// MajorComponents/FB_BPRequestor
(* BP Requestor
Elevates the BP request from an arbiter to PMPS_GVL.stRequestedBP
*)
FUNCTION_BLOCK FB_BPRequestor IMPLEMENTS I_HigherAuthority
VAR_INPUT
END_VAR
VAR_OUTPUT
    q_ReqBP : ST_BeamParams; // Arbitrated BP
END_VAR
VAR_IN_OUT
    Arbiter : FB_Arbiter;
    //FFO : FB_HardwareFFOutput;
END_VAR
VAR
    ReqBP : ST_BeamParams;
    nCohort : ULINT; // Current cohort, inc. 1 cycle after IO is updated
    nRequestCohort : ULINT; // Cohort number recorded at the time of the request.
END_VAR

Arbiter.ElevateRequest(THIS^); // Executes arbitration and retrieves ReqBP

IF nRequestCohort >= nCohort THEN
    // Update requested BP set
    q_ReqBP := ReqBP;
    // Note: we may do more here someday... perhaps all of the output control
    // will reside in here, and be solely controlled by this block. For now
    // I am going to adopt a flat management structure.
    // Start a new cohort
    nCohort := nCohort + 1;
END_IF

// Returns true when outputs to MPS are updated
METHOD CheckRequest : BOOL
VAR_INPUT
	nReqID	: DWORD;
END_VAR
VAR_INST
    xFirstTime : BOOL;
    nId : DWORD;
END_VAR
(* nRequestCohort will be < nCohort after output control
function blocks have been updated to reflect the new request
*)
CheckRequest := nRequestCohort < nCohort;
END_METHOD

METHOD RequestBP : BOOL
VAR_INPUT
	(*StateID of state requesting beam parameter set*)
	nReqID	: DWORD;
	(*Requested beam params*)
	stReqBP	: ST_BeamParams;
END_VAR
VAR_INST
    ReqID : DWORD;
    Registered : BOOL := FALSE;
END_VAR

// Check the request is coming from the same source we're used to
IF NOT Registered THEN
    ReqID := nReqID;
    Registered := TRUE;
END_IF
// log a complaint if false
RequestBP := ReqId = nReqId;

// Update internal BP request struct
ReqBP := stReqBP;

// Record current cohort

    nRequestCohort := nCohort;
END_METHOD

END_FUNCTION_BLOCK

// MajorComponents/FB_LinearGovernor

(* The governor is meant to check your work and keep you from making mistakes.

Checks:
Does your state match the device position and visa versa?
Are the beam parameters safe for the device state?
Did you properly assert the transition and final beam parameters?

*)
FUNCTION_BLOCK FB_LinearGovernor
VAR_INPUT
    i_stCurrentBeamParams    :    ST_BeamParams; //Link to global beam params
    i_xMPSOverride            :    BOOL; //True releases MPS limits after a delay
    i_xTransitionRequested    :    BOOL; //Set true to request a transition
    i_xResetMPSFault    :    BOOL; //Set true to clear MPS fault 
END_VAR
VAR_OUTPUT
     //True when governor has released restrictions
    q_xTransitionPermitted    :    BOOL;
    //Set if MC_Power has an error, or override mode is requested
    q_xFault    :    BOOL; 
    // Indicates override mode is active
    q_xMPSLimitsOverridden: BOOL;
END_VAR
VAR_IN_OUT
    stDevice    :    ST_Device; //The governed
    Arbiter    :    FB_Arbiter;
    FastFaultOutput    :    FB_HardwareFFOutput;
END_VAR
VAR
    mcPower    :    MC_Power;
    
    xActuatorPositiveEnable: BOOL;
    xActuatorNegativeEnable: BOOL;
    
    xMPSPositiveEnable    :    BOOL;
    xMPSNegativeEnable    :    BOOL;
    lrPosition: LREAL;
    
    lrLatchedTargetPosition    :    LREAL;
    lrLatchedTargetTolerance    :    LREAL;
    stLatchedTargetState    :    ST_DeviceStateExt;
    
    lrMPSUpperLimit: LREAL;
    lrMPSLowerLimit: LREAL;
    rtNewState: R_TRIG;
    xTransitionOK: BOOL;
    
    tonMPSOverrideMode    :    TON := (
        PT := T#5S
    );
    
    srMPSFault    :    SR;
    // Actuator out of bounds fault
    xActuatorOOB: BOOL;
    //Beam parameters out of spec
    xBeamParamsOOS: BOOL;
    //Beam parameters of currently latched state
    
    stLatchedBeamParams: ST_BeamParams;
    stTargetState: ST_DeviceStateExt;
    
    rtLatchNewState    :    R_TRIG;
    xInit: BOOL := TRUE;
    
    stInitDeviceState: ST_DeviceStateExt;
    // Indicates an error with initialization
    xInitFault: BOOL;
    // Indicates the state could not be found in the state table. There may be something wrong in the device state machine implementation or state table instantiation.
    xStateLookupError: BOOL;
    // A transition needs to be requested at least once before we start latching any state.
    xTransitionHasBeenRequested: BOOL := FALSE;
    ffBeamParamsOK : FB_FastFault;
    ffActuatorBoundsOK    :    FB_FastFault;
END_VAR


lrPosition := stDevice.stAxis.NcToPlc.ActPos; //Actuator position

stDevice.stAxis.ReadStatus();
//Init
(* The init strategy is:
If the device is restored and it's residing at the safe position,
no PMPS faults. *)
////////////////////////////////
    IF xInit THEN
        xInit := FALSE;
        //Use nSafeSate for initialization. 
        stDevice.StateTable.A_Lookup(key := stDevice.nSafeState);
        IF stDevice.StateTable.bOk THEN
            stInitDeviceState := F_DeviceState_To_DeviceStateExt(stDevice.StateTable.getValue, TRUE);
            xInitFault := FALSE;
        ELSE
            xInitFault := TRUE;
            stInitDeviceState.xValid := FALSE;
        END_IF
        lrLatchedTargetPosition := stInitDeviceState.rPosition;
        lrLatchedTargetTolerance := stInitDeviceState.rTolerance;
        stLatchedBeamParams := stInitDeviceState.stReqBeamParam;
    END_IF

// The governor will permit transitions once it verifies the transition assertion is active
// Note the governor does not verify the target state beam params are asserted, perhaps it should <TODO>
////////////////////////////////
    IF i_xTransitionRequested THEN
        xTransitionHasBeenRequested    := TRUE;
        
        xTransitionOK := Arbiter.CheckRequest( stDevice.stTransitionState.nStateRef) AND F_SafeBPCompare(i_stCurrentBeamParams, stDevice.stTransitionState.stReqBeamParam);
        
        //Set the target state for evaluation in further logic
        stdevice.StateTable.A_Lookup(key := stDevice.nTargetState);
        IF stDevice.StateTable.bOk THEN
            stTargetState := F_DeviceState_To_DeviceStateExt(stDevice.StateTable.getValue, TRUE);
            xStateLookupError := FALSE;
        ELSE
            xStateLookupError := TRUE;
            stTargetState.xValid := FALSE;
        END_IF
    ELSE
        xTransitionOK := FALSE;
    END_IF

(* Note about TransitionRequested

If TransitionRequested goes false during a transition, an MPS fault may be induced. This occurs
because the Actuator Out of Bounds fault will go back to using the original state limits, which
the axis may have already moved beyond.

To avoid this transient fault, make sure your device state machine is implemented such that the 
transition request to the governor block remains high until the target position is reached.
*)

//Determine if a transition is complete and latch the new state
(* A transition is complete when:

Axis at standstill.
Axis within tolerance.
No transition req.

Once these conditions are met, the MPS limits shall re-engage to restrict the
axis motion to the tolerance around the state position and the MPS fault monitors
shall evaluate based on the newly latched target state.
*)

rtLatchNewState(CLK := stDevice.stAxis.Status.StandStill AND
    lrPosition <= stTargetState.rPosition + stTargetState.rTolerance AND
    lrPosition >= stTargetState.rPosition - stTargetState.rTolerance AND
    NOT i_xTransitionRequested AND xTransitionHasBeenRequested);
    
IF rtLatchNewState.Q THEN
    lrLatchedTargetPosition := stTargetState.rPosition;
    lrLatchedTargetTolerance := stTargetState.rTolerance;
    stLatchedBeamParams := stTargetState.stReqBeamParam;
    stLatchedTargetState := stTargetState;
END_IF

//Let other blocks know the governor won't interfer with transitions
q_xTransitionPermitted := xTransitionOK;

//Adjust limit ranges based on active state and current target
IF xTransitionOK THEN
    //Extend range to include target state
    lrMPSUpperLimit := MAX(lrMPSUpperLimit, stTargetState.rPosition + stTargetState.rTolerance);
    lrMPSLowerLimit := MIN(lrMPSLowerLimit, stTargetState.rPosition - stTargetState.rTolerance);
ELSE
    //Calculate the limit positions for MPS based on current state
    lrMPSUpperLimit := lrLatchedTargetPosition + lrLatchedTargetTolerance;
    lrMPSLowerLimit := lrLatchedTargetPosition - lrLatchedTargetTolerance;
END_IF


//MPS override
(* In override mode, the device will be free to move anywhere within it's travel range *)
//Permit motion after a small delay
tonMPSOverrideMode(IN:=i_xMPSOverride OR stDevice.xOverrideMPSLimits, Q=>q_xMPSLimitsOverridden);

//Virtual limit switch evaluation
xActuatorPositiveEnable    := stDevice.i_xHiLim AND lrPosition <= stDevice.lrUpperPositionLimit;
xActuatorNegativeEnable    := stDevice.i_xLoLim AND lrPosition >= stDevice.lrLowerPositionLimit;

//Evaluate MPS limit states
xMPSPositiveEnable := lrPosition <= lrMPSUpperLimit;
xMPSNegativeEnable := lrPosition >= lrMPSLowerLimit;

//Final Limit switch evaluation
mcPower.Enable_Positive := xActuatorPositiveEnable AND (tonMPSOverrideMode.Q OR xMPSPositiveEnable);
mcPower.Enable_Negative := xActuatorNegativeEnable AND (tonMPSOverrideMode.Q OR xMPSNegativeEnable);

mcPower(
    Axis := stDevice.stAxis,
    Enable := stDevice.xEnable //link to device enable <TODO>
);



//MPS Faults
//Fault if the beam is unsafe for current state
ffBeamParamsOK(i_xOK:=F_SafeBPCompare(i_stCurrentBeamParams, stLatchedBeamParams), 
                i_xReset:=i_xResetMPSFault,
                io_fbFFHWO := FastFaultOutput);

//Fault if the position is outside of the permitted range
ffActuatorBoundsOK(i_xOK := (lrPosition <= lrMPSUpperLimit AND lrPosition >= lrMPSLowerLimit), 
                    i_xReset:=i_xResetMPSFault,
                io_fbFFHWO := FastFaultOutput);


    
//Collect all other faults
q_xFault := NOT ffBeamParamsOK.o_xFFLine OR
    NOT ffActuatorBoundsOK.o_xFFLine OR
    mcPower.Error    OR
    i_xMPSOverride    OR
    xInitFault;

//Any faults trip the fast fault line for this FB    
//FastFaultOutput.CheckIn(NOT q_xFault);

END_FUNCTION_BLOCK

// MajorComponents/FB_LRateFromEPICS
FUNCTION_BLOCK FB_LRateFromEPICS

(*
enum MPSBeamRates {
    MPSRateInvalid            =  0,
    MPSRate0Hz                =  1,
    /* Previously used 2 and 3 for single shot and burst */
    MPSRate1Hz                =  4,
    MPSRate10Hz               =  5,
    MPSRate30Hz               =  6,
    MPSRate60Hz               =  7,
    MPSRate120Hz              =  8,
    MPSRateUnknown            =  9,
    MPSRateSingleShot         = 10,
    MPSRateBurstMode          = 11,
    MPSRateBurstModeNotActive = 12,
    MPSNumberOfBeamRates      = 13,
    MPSRateBurstInvalid       = 14
}
*)

VAR_IN_OUT
	BP : ST_BeamParams;
END_VAR
VAR_OUTPUT
	xError : BOOL;
END_VAR
VAR
	{attribute 'pytmc' := '
        pv: L:Rate
        link: IOC:BSY0:MP01:BYKIK_RATE
        field: EGU RateEnum
    '}
    fbBYKIK_Rate : FB_LREALFromEPICS;
	
	eMPSRate : E_MPSBeamRates;
END_VAR
VAR CONSTANT
	cFailSafeRate : UINT := 120;
END_VAR

fbBYKIK_Rate();

eMPSRate := LREAL_TO_UINT(fbBYKIK_Rate.fValue);

CASE eMPSRate OF
	MPSRateInvalid:
		BP.nRate := cFailSafeRate;
	MPSRate0Hz:
		BP.nRate := 0;
	MPSRate1Hz:
		BP.nRate := 1;
	MPSRate10Hz:
		BP.nRate := 10;
	MPSRate30Hz:
		BP.nRate := 30;
	MPSRate60Hz:
		BP.nRate := 60;
	MPSRate120Hz:
		BP.nRate := 120;
	MPSRateUnknown:
		BP.nRate := cFailSafeRate;
	
ELSE
	BP.nRate := cFailSafeRate;
END_CASE

BP.xValid R= NOT fbBYKIK_Rate.bValid OR
			eMPSRate = MPSRateUnknown OR
			eMPSRate = MPSRateInvalid;

END_FUNCTION_BLOCK

// TestComponents/FB_Arbiter_Test
{attribute 'call_after_init'}
FUNCTION_BLOCK FB_Arbiter_Test EXTENDS TcUnit.FB_TestSuite
VAR_INPUT
END_VAR
VAR_OUTPUT
END_VAR
VAR
END_VAR

Arbitration();
RequestCheckRemoveBP();
FullArbitrationStack();

METHOD Arbitration
VAR_INPUT
END_VAR
VAR
    
     nTranReqID    :    UDINT    := 1;
    stAttReqBP    :    ST_BeamParams := PMPS_GVL.cstFullBeam;
    
    nPPEReqID    :    UDINT    := 2;
    stPPEReqBP    :    ST_BeamParams := PMPS_GVL.cstFullBeam;
    
    nEVReqID    :    UDINT    := 3;
    stEVReqBP    :    ST_BeamParams := PMPS_GVL.cstFullBeam;
    
    nRateReqID    :    UDINT    := 4;
    stRateReqBP    :    ST_BeamParams := PMPS_GVL.cstFullBeam;
    
    stArbitratedBP    :    ST_BeamParams;
    stExpectedBP    :    ST_BeamParams;
END_VAR
VAR_INST
    fbArbiter    :    FB_Arbiter(1);
END_VAR
TEST('Arbitration');

stAttReqBP.nTran := 50;
stPPEReqBP.fPP_mJ := 1;
stEVReqBP.neVRange := 2#1111_1100_1111_1111;
stRateReqBP.nRate := 10;

stExpectedBP.nTran     :=     stAttReqBP.nTran;
stExpectedBP.fPP_mJ    :=  stPPEReqBP.fPP_mJ;
stExpectedBP.neVRange := stEVReqBP.neVRange;
stExpectedBP.nRate := stRateReqBP.nRate;

//Load arbiter with beam parameter sets
AssertTrue(fbArbiter.AddRequest(nTranReqID, stAttReqBP),
                    'Safest attenuation request failed to load');
                    
//Load arbiter with beam parameter sets
AssertTrue(fbArbiter.AddRequest(nPPEReqID, stPPEReqBP),
                    'Safest PPE request failed to load');
                    
//Load arbiter with beam parameter sets
AssertTrue(fbArbiter.AddRequest(nEVReqID, stEVReqBP),
                    'Safest stEVReqBP request failed to load');
                    
//Load arbiter with beam parameter sets
AssertTrue(fbArbiter.AddRequest(nRateReqID, stRateReqBP),
                    'Safest stRateReqBP request failed to load');

stArbitratedBP := fbArbiter.GetArbitratedBP();

AssertFalse(F_DifferentBeamParams(stExpectedBP, stArbitratedBP),
                'Arbitrated BP does not match expected.');

TEST_FINISHED();
END_METHOD

METHOD FullArbitrationStack
VAR_INPUT
END_VAR
VAR   
    nId    :    DWORD := 1;
    stReq    :    ST_BeamParams := (nTran:=12);
END_VAR
VAR_INST
    fbArbiter    :    FB_Arbiter(1);
    
    fbHigherArb : FB_Arbiter(2);
    
    fbSubSysToArb : FB_SubSysToArbiter_IO; // Subsystem interface with beamline arbiter PLC
    pBPR : POINTER TO ST_BeamParams_IO;
    
    fbArbToSubSys : FB_ArbiterToSubSys_IO := (RequestingSystemID:=42); // Beamline arbiter PLC interface with subsystems
    pBPC : POINTER TO ST_BeamParams_IO;
    
    fbBPR : FB_BPRequestor; // Use in the arbiter PLC to apply an arbitrated beam parameter set to the accelerator interface
    
    FFO : FB_HardwareFFOutput; // Dummy FFO not important for these tests

    Cycle : INT := 0;
    
    CycleLimit : INT := 20;
    
END_VAR
VAR CONSTANT
    SysID : DWORD := 42;
END_VAR
// This simulates a synchronous cycle between the subsystem and arbiter PLC cycles. Ie. phase is locked, and cycle time is the same. This is not always the case, so these tests should be 
// trusted with a grain of salt.

TEST('FullStack');



CASE Cycle OF

0: 
    IF NOT fbArbiter.CheckRequestInPool(nID) THEN
        AssertTrue(fbArbiter.AddRequest(nId, stReq), 'Arbiter returned false from AddRequest'); // some device asking its local arbiter for some beam parameters
    END_IF  
    
    TEST('JustEnteredRequest');
    AssertFalse(fbArbiter.CheckRequest(nId),
        'Check should fail. Request not arbitrated yet.');
    TEST_FINISHED();
   
8000:
    TEST_FINISHED_NAMED('FullStack');   
    
END_CASE 


TEST('VerifyBPRHasBP');
IF fbHigherArb.CheckRequest(SysID) THEN
    AssertFalse(F_DifferentBeamParams(stReq, fbBPR.q_ReqBP),
        'Beam parameters not fully propagated to BPR at highest level');
        TEST_FINISHED_NAMED('VerifyBPRHasBP');
END_IF

TEST('ArbToSubsysPropagation');
IF fbArbToSubSys.nActiveCohort = fbArbToSubSys.nRequestedCohort 
    AND fbArbToSubSys.nActiveCohort <> 0 THEN
    AssertTrue(fbHigherArb.CheckRequest(SysID),
        'Active cohort = Requested cohort before higher arbiter confirmed request was active');
    TEST_FINISHED_NAMED('ArbToSubsysPropagation');
END_IF

TEST('SubsysToArbPropagation');
IF fbArbiter.CheckRequest(nId) THEN
    AssertTrue(fbSubSysToArb.nActiveCohort >= fbSubSysToArb.nRequestCohort,
        'Request validated before higher level confirmation');
    TEST_FINISHED_NAMED('SubsysToArbPropagation');
END_IF


TEST('VerifyIncludedAtAllLevels');
IF fbArbiter.CheckRequest(nId) THEN
    AssertTrue(fbHigherArb.xActiveInArbitration, 'HigherArb is not yet included in arbitration');
    AssertTrue(fbArbiter.xActiveInArbitration, 'Local Arb is not yet included in arbitration');
    TEST_FINISHED_NAMED('VerifyIncludedAtAllLevels');
END_IF
      
    
///////////////////////////////////////
//Sub system cycle
fbSubSysToArb(Arbiter := fbArbiter, fbFFHWO := FFO);
//END of sub system cycle
///////////////////////////////////////

//Ethercat transfer simulation
// Transfer of requested BP to arbiter PLC
pBPR := ADR(fbArbToSubSys.i_RequestedBP);
pBPR^ := fbSubSysToArb.q_stRequestedBP;

// Transfer of current BP to sub system PLC
pBPC := ADR(fbSubSysToArb.i_stCurrentBP);
pBPC^ := fbArbToSubSys.o_CurrentBP;

//////////////////////////////////////
//Start of arbiter plc cycle
//Arb io collects sub system status
fbArbToSubSys(Arbiter := fbHigherArb, fbFFHWO := FFO); // This is making a request in the higher arb
//BPR collects arbiter summation
fbBPR(Arbiter := fbHigherArb); // This is getting the arbitrated BP




IF CycleLimit > Cycle THEN
    Cycle := Cycle + 1;
ELSE 
    Cycle := 8000;
END_IF
END_METHOD

METHOD RequestCheckRemoveBP
VAR_INPUT
END_VAR
VAR
    
    nId    :    DWORD := 1;
    stReq    :    ST_BeamParams;
END_VAR
VAR_INST
    fbArbiter    :    FB_Arbiter(1);
END_VAR
TEST('RequestBP');
AssertTrue(fbArbiter.AddRequest(nId, stReq),
    'Request failed');

TEST_FINISHED();
    
TEST('DuplicateID');
AssertFalse(fbArbiter.AddRequest(nId, stReq),
    'Duplicate request accepted, not good.');

TEST_FINISHED();
    
TEST('CheckBP');
AssertFalse(fbArbiter.CheckRequest(nId),
    'Check should fail. Request not arbitrated yet.');
TEST_FINISHED();

TEST('CheckBPArbitrated');
WRITE_PROTECTED_ULINT(ADR(fbArbiter.nArbiterCohort), fbArbiter.nArbiterCohort + 1);
WRITE_PROTECTED_BOOL(ADR(fbArbiter.xActiveInArbitration), TRUE);
AssertTrue(fbArbiter.CheckRequest(nId),
    'Check should pass.');

TEST_FINISHED();      
    
TEST('IDDoesNotExist');
WRITE_PROTECTED_ULINT(ADR(fbArbiter.nArbiterCohort), fbArbiter.nArbiterCohort + 1); 
AssertFalse(fbArbiter.CheckRequest(nId+1),
    'Check returned true when ID does not exist');

TEST_FINISHED();
    
TEST('RemoveBP');
AssertTrue(fbArbiter.RemoveRequest(nId),
    'Remove failed');
AssertFalse(fbArbiter.CheckRequest(nId),
    'Remove did not remove request');
    
TEST_FINISHED();
END_METHOD

END_FUNCTION_BLOCK

// TestComponents/FB_ArbToSubsys_Test
{attribute 'call_after_init'}
FUNCTION_BLOCK FB_ArbToSubsys_Test EXTENDS TcUnit.FB_TestSuite
VAR_INPUT
END_VAR
VAR_OUTPUT
END_VAR
VAR
END_VAR

BasicFunction();

METHOD BasicFunction
VAR_INPUT
END_VAR
VAR CONSTANT
    SysID : DWORD := 42;
END_VAR
VAR   
    nId    :    DWORD := 1;
    stReq    :    ST_BeamParams := (nTran:=12);
END_VAR
VAR_INST
    fbArbiter    :    FB_Arbiter(1);
    
    pBPR : POINTER TO ST_BeamParams_IO;
    
    stBPRIO : ST_BeamParams_IO := (
        nCohortInt := 1,
        nTran := 35); // Simulates subsystem BP request
    
    fbArbToSubSys : FB_ArbiterToSubSys_IO := (RequestingSystemID:=42); // Beamline arbiter PLC interface with subsystems
    pBPC : POINTER TO ST_BeamParams_IO;
    
    fbBPR : FB_BPRequestor; // Use in the arbiter PLC to apply an arbitrated beam parameter set to the accelerator interface
    
    FFO : FB_HardwareFFOutput; // Dummy FFO not important for these tests

    Cycle : INT := 0;
    
    CycleLimit : INT := 20;
    
END_VAR

// Simulate an initial cycle with no new requests coming in
fbArbToSubSys(Arbiter:=fbArbiter, fbFFHWO:=FFO);

TEST('Init');
TEST_FINISHED();

//Ethercat transfer simulation
// Transfer of requested BP to arbiter PLC
pBPR := ADR(fbArbToSubSys.i_RequestedBP);
pBPR^ := stBPRIO;

///////////////////////////////////////
//Sub system cycle
fbArbToSubSys(Arbiter:=fbArbiter, fbFFHWO:=FFO);
//END of sub system cycle
///////////////////////////////////////


TEST('New request');
    AssertTrue(fbArbToSubSys.nRequestedCohort = fbArbToSubSys.i_RequestedBP.nCohortInt, 'ReqCohort and qBP Cohort do not match, and they should');
    AssertTrue(fbArbiter.CheckRequestInPool(SysID), 'ArbToSubSys request should be in arbiter pool now');
    AssertTrue(fbArbToSubSys.nActiveCohort = 0, 'Active cohort should remain the initial value until the current request is active in higher arbitration');
    AssertTrue(fbArbToSubSys.o_CurrentBP.nCohortInt = fbArbToSubSys.nActiveCohort, 'Cohort being sent to sub system remains unincremented');
TEST_FINISHED_NAMED('New request');
    

///////////////////////////////////////
//Sub system cycle
fbBPR(Arbiter:=fbArbiter);
fbArbToSubSys(Arbiter:=fbArbiter, fbFFHWO:=FFO);
//END of sub system cycle
///////////////////////////////////////

///////////////////////////////////////
//Sub system cycle
fbBPR(Arbiter:=fbArbiter);
fbArbToSubSys(Arbiter:=fbArbiter, fbFFHWO:=FFO);
//END of sub system cycle
///////////////////////////////////////


TEST('Request has become active');
    AssertTrue(fbArbToSubSys.nRequestedCohort = fbArbToSubSys.nActiveCohort, 'ReqCohort and qBP Cohort do not match, and they should');
    AssertTrue(fbArbiter.CheckRequest(SysID), 'ArbToSubSys request should be in arbiter pool now');
    AssertTrue(fbArbToSubSys.nActiveCohort = stBPRIO.nCohortInt, 'Active cohort should remain the initial value until the current request is active in higher arbitration');
    AssertTrue(fbBPR.q_ReqBP.nTran = stBPRIO.nTran, 'BPR and requested BP should match');
TEST_FINISHED_NAMED('Request has become active');
END_METHOD

END_FUNCTION_BLOCK

// TestComponents/FB_AttenuatorSimulator
FUNCTION_BLOCK FB_AttenuatorSimulator
VAR_INPUT
    i_rRequestedAttenuation    :    REAL;
    i_stBPReadback    :    ST_BeamParams;
END_VAR
VAR_OUTPUT
    q_xFault    :    BOOL;
    q_rCurrentAttenuation    :    REAL;
END_VAR
VAR_IN_OUT
    Arbiter    :    FB_Arbiter; //Higher level arbiter from which upstream attenuation can be requested
END_VAR
VAR
    tonDelay    :    TON := (
        PT := T#3S
        );
END_VAR

// Really basic delay
tonDelay(IN := i_rRequestedAttenuation <> q_rCurrentAttenuation);

IF tonDelay.Q THEN
    q_rCurrentAttenuation := i_rRequestedAttenuation;
END_IF

END_FUNCTION_BLOCK

// TestComponents/FB_BPTM_Test
{attribute 'call_after_init'}
FUNCTION_BLOCK FB_BPTM_Test EXTENDS TcUnit.FB_TestSuite
VAR_INPUT
END_VAR
VAR_OUTPUT
END_VAR
VAR
END_VAR

BPTMBasicFunction();

METHOD BPTMBasicFunction
VAR_INPUT
END_VAR
VAR    
    //Final and transition assertions
    nTransitionID    :    UDINT := 1;
    stTransitionAssertion    :    ST_BeamParams := PMPS_GVL.cstSafeBeam;
    
     nReqID    :    UDINT    := 2;
    stReqAssertion    :    ST_BeamParams := PMPS_GVL.cstSafeBeam;
    
    fbMachine    :    FB_MachineSimulator;    
    
END_VAR
VAR_INST
    fbBPTM_TestBasicFunction    :    BeamParameterTransitionManager;
    fbArbiter    :    FB_Arbiter(1);
    fbBPR :  FB_BPRequestor;
    xFirstPass    :    BOOL := TRUE;
    eTestStep: eBPTMTestStates := eBPTMTestStates.Init;
END_VAR
CASE eTestStep OF

eBPTMTestStates.Init:
    
    TEST('BPTMTest');
    eTestStep := eBPTMTestStates.WaitingForTransitionAssertion;

eBPTMTestStates.WaitingForTransitionAssertion:
    TEST('BPTM Requests Transition');
    
    //Call BPTM with requested final state and transition state
    fbBPTM_TestBasicFunction(
        fbArbiter := fbArbiter,
        i_TransitionAssertionID := nTransitionID,
        i_stTransitionAssertion := stTransitionAssertion,
        
        i_nRequestedAssertionID := nReqID,
        i_stRequestedAssertion := stReqAssertion
    );
    
    IF fbBPTM_TestBasicFunction.eBPTMState = E_BPTMState.WaitingForTransitionAssertion AND 
        NOT fbBPTM_TestBasicFunction.xEntry THEN
    
        AssertTrue(fbArbiter.CheckRequestInPool(nTransitionID), 'Arbiter did not accept BPTM transition assertion');
        
        AssertFalse(fbArbiter.CheckRequestInPool(nReqID), 'BPTM has requested final too early.');
                
        AssertFalse(fbBPTM_TestBasicFunction.q_xTransitionAuthorized,
            'Transition should not be authorized until the arbiter has final assertion');
            
        TEST_FINISHED_NAMED('BPTM Requests Transition');
        
        eTestStep := eBPTMTestStates.WaitingForFinalAssertion;
    END_IF

eBPTMTestStates.WaitingForFinalAssertion:

    TEST('BPTM Requests Final');
    fbBPTM_TestBasicFunction(fbArbiter := fbArbiter,
        stCurrentBeamParameters := stTransitionAssertion);
    
    IF fbBPTM_TestBasicFunction.eBPTMState = E_BPTMState.WaitingForFinalAssertion AND
        NOT fbBPTM_TestBasicFunction.xEntry THEN
    
        AssertTrue(fbArbiter.CheckRequest(nTransitionID), 
            'Transition assertion should be active in arbitration now.');
        
        AssertTrue(fbArbiter.CheckRequestInPool(nReqID),
            'Final assertion should be in arbiter');
            
        AssertFalse(fbBPTM_TestBasicFunction.q_xTransitionAuthorized,
            'Transition should not be authorized until the final request is active in arbitration');
            
        TEST_FINISHED_NAMED('BPTM Requests Final');
   
        eTestStep := eBPTMTestStates.Transitioning;
    END_IF

eBPTMTestStates.Transitioning:
    TEST('BPTM Authorizes Transition');
    fbBPTM_TestBasicFunction(fbArbiter := fbArbiter,
        stCurrentBeamParameters := stTransitionAssertion);
        
    IF fbBPTM_TestBasicFunction.eBPTMState = E_BPTMState.Transitioning AND
        NOT fbBPTM_TestBasicFunction.xEntry THEN
    
        AssertTrue(fbArbiter.CheckRequest(nReqID),
            'Transition assertion should be in arbiter');
        
        AssertTrue(fbArbiter.CheckRequest(nReqID),
            'Final assertion should be in arbiter');
            
        AssertTrue(fbBPTM_TestBasicFunction.q_xTransitionAuthorized,
            'Transition should be authorized at this point.');
            
        AssertEquals(nReqID, fbBPTM_TestBasicFunction.nCurrentAssertionID,
            'nCurrentAssertionID not set.');
    
        TEST_FINISHED_NAMED('BPTM Authorizes Transition');
        
        eTestStep := eBPTMTestStates.CleaningUp;
    END_IF

eBPTMTestStates.CleaningUp:
    TEST_FINISHED_NAMED('BPTMTest');    
    
END_CASE

// Completes arbiter request elevation process
// Necessary for CheckRequest to return true, ever
fbBPR(Arbiter:=fbArbiter);
END_METHOD

END_FUNCTION_BLOCK

// TestComponents/FB_DiffBP_Test
{attribute 'call_after_init'}
FUNCTION_BLOCK FB_DiffBP_Test EXTENDS TcUnit.FB_TestSuite
VAR_INPUT
END_VAR
VAR_OUTPUT
END_VAR
VAR

END_VAR


BPDiff();

//Verify BP comparison remains logical.
METHOD BPDiff
VAR_INPUT
END_VAR
VAR
    BP1    :    ST_BeamParams;
    BP2    :    ST_BeamParams;
END_VAR
TEST('BPDiffCheck');

BP2.nTran := 10; 
    
AssertTrue(
    F_DifferentBeamParams(BP1, BP2),
    'DifferentBP eval is broken (True)'); 

BP1.nTran := BP2.nTran;   
    
AssertFalse(
    F_DifferentBeamParams(BP2, BP1),
    'DifferentBP eval is broken (False)');

TEST_FINISHED();
END_METHOD

END_FUNCTION_BLOCK

// TestComponents/FB_evRangeCalculator_Test
{attribute 'call_after_init'}
FUNCTION_BLOCK FB_evRangeCalculator_Test EXTENDS FB_TestSuite
VAR_INPUT
END_VAR
VAR_OUTPUT
END_VAR
VAR
END_VAR

BasicFunction();

METHOD BasicFunction
VAR_INPUT
END_VAR
VAR
    {attribute 'displaymode' := 'binary'}
    LastWord : WORD := 2#0000_0000_0000_0010;
    {attribute 'displaymode' := 'binary'}
    Result : WORD;
    {attribute 'displaymode' := 'binary'}
    TestEV : WORD;
    
    {attribute 'displaymode' := 'binary'}
    tEvW : WORD;
    tEv : REAL;
    
    
    fbStr : FB_FormatString;
END_VAR
VAR CONSTANT
    nLowerLimitBoundary : INT := 0;
END_VAR
Test('CheckRanges');

//Lower limit equal
tEvW.nLowerLimitBoundary := TRUE;
tEv := PMPS_GVL.g_areVBoundaries[nLowerLimitBoundary];
Result := F_eVRangeCalculator(tEv, 0);
AssertTrue(
    Result = tEvW,
    'Lower limit not inclusive');
//Mid range
AssertTrue(
    F_eVRangeCalculator(251, 0) = 2#0000_0000_0000_0010,
    'In range failed, whatever you did, it broke this really bad.');
//Out of range
AssertFalse(
    F_eVRangeCalculator(301, 0) = 2#0000_0000_0000_0010,
    'Out of range failed, whatever you did, it broke this really bad.');

TEST_FINISHED();

Test('Negative eV failsafes');
//Negative eV
AssertTrue(
    F_eVRangeCalculator(-300, 0) = 16#FFFF,
    'Working with antimatter? Negative eV should failsafe to FFFF.');    

TEST_FINISHED();

Test('Check hyst keeps');

LastWord := F_eVRangeCalculator(250, 2#0000_0000_0000_0000);

AssertTrue(
    F_eVRangeCalculator(304, 2#0000_0000_0000_0010) = 2#0000_0000_0000_0110,
    'Moving up does not stick.');
    
    Result := F_eVRangeCalculator(196, 2#0000_0000_0000_0010);
    TestEV := 2#0000_0000_0000_0011;
    fbStr.arg1 := F_WORD(Result);
    fbStr.arg2 := F_WORD(TestEV);
    fbStr.sFormat := 'Moving down does not stick. Result: %b vs. Test: %b';
    fbStr();
    
AssertTrue(Result = TestEV,
    fbStr.sOut);

TEST_FINISHED();

Test('Check hyst drops');

AssertTrue(
    F_eVRangeCalculator(351, 2#0000_0000_0000_0010) = 2#0000_0000_0000_0100,
    'Moving up does not drop.');
    
AssertTrue(
    F_eVRangeCalculator(149, 2#0000_0000_0000_0010) = 2#0000_0000_0000_0001,
    'Moving down does not drop.');

TEST_FINISHED();
END_METHOD

END_FUNCTION_BLOCK

// TestComponents/FB_eVWithinSpec_Test
{attribute 'call_after_init'}
FUNCTION_BLOCK FB_eVWithinSpec_Test EXTENDS TcUnit.FB_TestSuite
VAR_INPUT
END_VAR
VAR_OUTPUT
END_VAR
VAR
END_VAR

evWithinRangeChecks();

METHOD evWithinRangeChecks
VAR_INPUT
END_VAR
VAR

END_VAR
TEST('evWithinRangeChecks');
    
//Upper limit equal
AssertTrue(
    F_eVWithinSpec(300, 2#0000_0000_0000_0010),
    'Upper limit not inclusive');
//Lower limit equal
AssertTrue(
    F_eVWithinSpec(300, 2#0000_0000_0000_0100),
    'Lower limit not inclusive');
//Out of range
AssertFalse(
    F_eVWithinSpec(300.1, 2#0000_0000_0000_0010),
    'Out of range failed, whatever you did, it broke this really bad.');
//Negative eV
AssertFalse(
    F_eVWithinSpec(-300, 16#FFFF),
    'Working with antimatter? Negative eV should not be acceptable.');
//Upper unallocated range
AssertFalse(
    F_eVWithinSpec(1701, 2#1000_0000_0000_0000),
    'eV range should not evaluate past 1.7keV');
    
TEST_FINISHED();
END_METHOD

END_FUNCTION_BLOCK

// TestComponents/FB_FastFault_Test
{attribute 'call_after_init'}
FUNCTION_BLOCK FB_FastFault_Test EXTENDS TcUnit.FB_TestSuite
VAR_INPUT
END_VAR
VAR_OUTPUT
END_VAR
VAR

END_VAR

FFCombinedFunctionality();
FFRegistration();

METHOD FFCombinedFunctionality
VAR_INPUT
END_VAR
VAR_INST
    fbFF    :    FB_FastFault;
    fbFFO    :    FB_HardwareFFOutput;
    
END_VAR
TEST('FFCombinedFunctionality');

//Clear initial faults
fbFFO.i_xReset:=TRUE; //Reset requested at start of cycle

fbFF(io_fbFFHWO := fbFFO, //FF reset somehwere in code
    i_xOK := TRUE,
    i_xReset := TRUE);

fbFFO.EvaluateOutput(); //FFO eval called at end of cycle
    
AssertTrue(fbFFO.q_xFastFaultOut,
    'Fast fault did not clear');


//Induce fault with FF

fbFFO(i_xReset := FALSE); //Reset released at start of cycle

fbFF(io_fbFFHWO := fbFFO, //FF faulted
    i_xOK := FALSE); //Reset is still set true from last call.
    
fbFFO.EvaluateOutput(); //FFO eval called at end of cycle

AssertFalse(fbFFO.q_xFastFaultOut,
    'Fast fault did not trip the beam');
    
    
//FFO remains faulted until local (FF) and FFO receieve fresh reset request, and faults
//are actually cleared

//Attempt to clear FFO fails because FF still faulted
fbFFO.i_xReset := TRUE; //Reset requested

fbFF(io_fbFFHWO := fbFFO, //FF faulted
    i_xOK := FALSE,
    i_xReset := FALSE);
    
fbFFO.EvaluateOutput(); //FFO eval called at end of cycle

AssertFalse(fbFFO.q_xFastFaultOut,
    'Fast fault output cleared while fault remains, very bad');
    
//Attempt to clear FF while fault remains fails
fbFFO.EvaluateOutput(i_xReset := FALSE);

fbFFO.i_xReset := TRUE; //Reset requested

fbFF(io_fbFFHWO := fbFFO, //FF faulted
    i_xOK := FALSE,
    i_xReset := TRUE); //This reset should fail.
    
fbFFO.EvaluateOutput(); //FFO eval called at end of cycle

AssertFalse(fbFFO.q_xFastFaultOut,
    'Fast fault cleared while fault remains, very bad');
    
TEST_FINISHED();
END_METHOD

METHOD FFRegistration
VAR_INPUT
END_VAR
VAR_INST
    fbFF    :    FB_FastFault;
    fbFFO    :    FB_HardwareFFOutput;
    astFF : ARRAY[0..10] OF ST_FF;
END_VAR
TEST('FFRegistration');

fbFF(io_fbFFHWO := fbFFO);

AssertEquals_STRING(fbFF.sPath, fbFFO.astFF[fbFF.RegistrationIdx].Info.sPath,
    'FF registration with FFO did not succeed');

TEST_FINISHED();
END_METHOD

END_FUNCTION_BLOCK

// TestComponents/FB_PhotonEnergyWatcher_Test
{attribute 'call_after_init'}
FUNCTION_BLOCK FB_PhotonEnergyWatcher_Test EXTENDS TcUnit.FB_TestSuite
VAR_INPUT
END_VAR
VAR_OUTPUT
END_VAR
VAR

END_VAR

PEWatcherBasicFunction();

METHOD PEWatcherBasicFunction
VAR_INPUT
END_VAR
VAR_INST
    fbPEW    :    FB_PhotonEnergyWatcher;
    fbFFO    :    FB_HardwareFFOutput;
    q_Output    :    BOOL;
    
    stCurBeamParams    :    ST_BeamParams;
    stMachineTargetBeamParams    :    ST_BeamParams;
    stReqBeamParams    :    ST_BeamParams;
END_VAR
TEST('PEWatcherBasicFunction');

//Clear FFO fault to start
fbFFO(i_xReset:=TRUE);

//All eV OK
stCurBeamParams.neVRange := F_eVRangeCalculator(800, 0);
    
stMachineTargetBeamParams.neVRange := 2#0000_0000_1000_0000;

stReqBeamParams.neVRange := 2#1111_1111_1111_1111;    

fbFFO(i_xReset:=FALSE); //Reset request released
    
fbPEW(i_stCurrentBeamParams := stCurBeamParams,
    i_stMachineTargetBeamParams := stMachineTargetBeamParams,
    i_stRequestedBeamParams := stReqBeamParams,
    io_fbFFHWO := fbFFO,
    i_xReset := TRUE); //Clear local FF within PEW
    
fbFFO.EvaluateOutput(q_xFastFaultOut=>q_Output); //This simulates a completed PLC cycle
//Evaluate output should be called once at the end of a PLC cycle.

AssertTrue(q_Output,
    'Beam within limits, FFO should be true');
    
    
//Req eV moved out of range
stCurBeamParams.neVRange := F_eVRangeCalculator(800, 0);
    
stMachineTargetBeamParams.neVRange := F_eVRangeCalculator(800, 0);

stReqBeamParams.neVRange := 2#0000_1111_0011_1111;

fbPEW.i_xReset := FALSE; //release local FF reset req    
fbPEW(i_stCurrentBeamParams := stCurBeamParams,
    i_stMachineTargetBeamParams := stMachineTargetBeamParams,
    i_stRequestedBeamParams := stReqBeamParams,
    io_fbFFHWO := fbFFO);
    
fbFFO.EvaluateOutput(q_xFastFaultOut=>q_Output);

AssertFalse(q_Output,
    'Limits moved beyond current and target beam, should produce a fault.');

//Beam and target eV moved back within permitted ranges, reset clears fault
stCurBeamParams.neVRange := F_eVRangeCalculator( 300, 0);
    
stMachineTargetBeamParams.neVRange := F_eVRangeCalculator(300, 0);

stReqBeamParams.neVRange := 2#0000_1111_0011_1111;

fbFFO(i_xReset:=TRUE); //New reset request

fbPEW.i_xReset := TRUE; //New reset request

fbPEW(i_stCurrentBeamParams := stCurBeamParams, //Beam params are now within spec
    i_stMachineTargetBeamParams := stMachineTargetBeamParams,
    i_stRequestedBeamParams := stReqBeamParams,
    io_fbFFHWO := fbFFO);
    
fbFFO.EvaluateOutput(q_xFastFaultOut=>q_Output);

AssertTrue(q_Output,
    'Beam within limits after reset, FFO should be true');
    
//At this point, the fast fault would be cleared

//Current beam eV moved out of range
stCurBeamParams.neVRange := F_eVRangeCalculator(800, 0); //Moved out of range
    
stMachineTargetBeamParams.neVRange := F_eVRangeCalculator(300, 0); //Still within range

stReqBeamParams.neVRange := 2#0000_1111_0011_1111;

fbPEW(i_stCurrentBeamParams := stCurBeamParams,
    i_stMachineTargetBeamParams := stMachineTargetBeamParams,
    i_stRequestedBeamParams := stReqBeamParams,
    io_fbFFHWO := fbFFO);
    
fbFFO.EvaluateOutput(q_xFastFaultOut=>q_Output);

AssertFalse(q_Output,
    'Current beam moved beyond set limits, should produce a fault');

//Target beam eV moved out of range
fbFFO(i_xReset:=FALSE); //Reset released
fbFFO(i_xReset:=TRUE); //New reset request comes in at the top of a cycle, but will be overridden

stCurBeamParams.neVRange := F_eVRangeCalculator(300, 0); //Now within range
    
stMachineTargetBeamParams.neVRange := F_eVRangeCalculator(800, 0); //Moved out of range

stReqBeamParams.neVRange := 2#0000_1111_0011_1111;

fbPEW.i_xReset := TRUE; //Attempt to reset local FF will fail
fbPEW(i_stCurrentBeamParams := stCurBeamParams,
    i_stMachineTargetBeamParams := stMachineTargetBeamParams,
    i_stRequestedBeamParams := stReqBeamParams,
    io_fbFFHWO := fbFFO);
    
fbFFO.EvaluateOutput(q_xFastFaultOut=>q_Output);

AssertFalse(q_Output,
    'Target beam moved beyond set limits, should produce a fault');
    
TEST_FINISHED();
END_METHOD

END_FUNCTION_BLOCK

// TestComponents/FB_SafeBPCompare_Test
{attribute 'call_after_init'}
FUNCTION_BLOCK FB_SafeBPCompare_Test EXTENDS TcUnit.FB_TestSuite
VAR_INPUT
END_VAR
VAR_OUTPUT
END_VAR
VAR

END_VAR

BeamOffIsSafe();
BPComparisonCheck();

//Verify beam off is considered safe.
METHOD BeamOffIsSafe
VAR_INPUT
END_VAR
VAR
    stBeamOn_MoreConservative    :    ST_BeamParams;
    stBeamOff_LessConservative    :    ST_BeamParams;
END_VAR
stBeamOn_MoreConservative  := F_SetBeamParams(
    50, //50% attenuation is more conservative than 0
    10,
    16#FFFF,
    120, //rate
    PMPS_GVL.DUMMY_AUX_ATT_ARRAY);

stBeamOff_LessConservative:= F_SetBeamParams(
    0, //0% attenuation, less conservative, without 0-rate this beam parameter set would be less safe than above
    10,
    16#FFFF,
    0, //rate, hence, more conservative
    PMPS_GVL.DUMMY_AUX_ATT_ARRAY); //0 beam rate means this bps is actually safer than BeamOn

TEST('BeamOffIsSafe');
    
AssertTrue(
    F_SafeBPCompare(stBeamOff_LessConservative, stBeamOn_MoreConservative),
    'SafeBPCompare does not think beam rate = 0 is safer than anything else.'); 
TEST_FINISHED();
END_METHOD

//Verify BP comparison remains logical.
METHOD BPComparisonCheck
VAR_INPUT
END_VAR
VAR
    stSafer    :    ST_BeamParams;
    stNotSoSafe    :    ST_BeamParams;
    idx : UINT;
END_VAR


TEST('BPComparisonTran');
//Attenuation
stSafer := F_SetBeamParams(
    0, //
    10,
    16#FFFF,
    1,
    PMPS_GVL.DUMMY_AUX_ATT_ARRAY);

stNotSoSafe := F_SetBeamParams(
    1, //
    10,
    16#FFFF,
    1,
    PMPS_GVL.DUMMY_AUX_ATT_ARRAY); 
    
AssertTrue(
    F_SafeBPCompare(stSafer, stNotSoSafe),
    'Attenuation eval is broken (True)'); 

AssertFalse(
    F_SafeBPCompare(stNotSoSafe, stSafer),
    'Attenuation eval is broken (False)');

TEST_FINISHED();
    
//Attenuator array    
TEST('BPComparisonTranArray');

stNotSoSafe := F_SetBeamParams(
    0, //
    10,
    16#FFFF,
    1,
    PMPS_GVL.DUMMY_AUX_ATT_ARRAY); 

FOR idx:=1 TO PMPS_GVL.AUX_ATTENUATORS DO
    stSafer.astAttenuators[idx].nTran := 30;
    stNotSoSafe.astAttenuators[idx].nTran := 50;
    
    AssertTrue(
    F_SafeBPCompare(stSafer, stNotSoSafe),
    'Attenuation array eval is broken (True)'); 

    AssertFalse(
    F_SafeBPCompare(stNotSoSafe, stSafer),
    'Attenuation array eval is broken (False)');
    
    IF NOT F_SafeBPCompare(stSafer, stNotSoSafe) or F_SafeBPCompare(stNotSoSafe, stSafer) THEN
        EXIT; // Exit this loop on the first failure.
	END_IF
    
    stSafer.astAttenuators[idx].nTran := 0;
    stNotSoSafe.astAttenuators[idx].nTran := 0;
    
END_FOR

TEST_FINISHED();

stSafer.astAttenuators[idx].nTran := 0;
stNotSoSafe.astAttenuators[idx].nTran := 0;

//Aperture array
TEST('BPComparisonApertureArray');

FOR idx:=1 TO PMPS_GVL.MAX_APERTURES DO
    // Height
    stSafer.astApertures[idx].Height := 30; // narrower is safer
    stNotSoSafe.astApertures[idx].Height := 50;
    
    AssertTrue(
    F_SafeBPCompare(stSafer, stNotSoSafe),
    'Aperture array eval is broken on height (True)'); 

    AssertFalse(
    F_SafeBPCompare(stNotSoSafe, stSafer),
    'Aperture array eval is broken on height (False)');
    
    IF NOT F_SafeBPCompare(stSafer, stNotSoSafe) or F_SafeBPCompare(stNotSoSafe, stSafer) THEN
        EXIT; // Exit this loop on the first failure.
	END_IF
    
    stSafer.astApertures[idx].Height := 0;
    stNotSoSafe.astApertures[idx].Height := 0;
    
    // Width
    stSafer.astApertures[idx].Width := 30; // narrower is safer
    stNotSoSafe.astApertures[idx].Width := 50;
    
    AssertTrue(
    F_SafeBPCompare(stSafer, stNotSoSafe),
    'Aperture array eval is broken on width (True)'); 

    AssertFalse(
    F_SafeBPCompare(stNotSoSafe, stSafer),
    'Aperture array eval is broken on width (False)');
    
    IF NOT F_SafeBPCompare(stSafer, stNotSoSafe) or F_SafeBPCompare(stNotSoSafe, stSafer) THEN
        EXIT; // Exit this loop on the first failure.
	END_IF
    
    stSafer.astApertures[idx].Width := 0;
    stNotSoSafe.astApertures[idx].Width := 0;
    
    
END_FOR

TEST_FINISHED();
    
//Rate
TEST('BPComparisonRate');
stSafer := F_SetBeamParams(
    0,
    10,
    16#FFFF,
    1,
    PMPS_GVL.DUMMY_AUX_ATT_ARRAY); //

stNotSoSafe := F_SetBeamParams(
    0,
    10,
    16#FFFF,
    10,
    PMPS_GVL.DUMMY_AUX_ATT_ARRAY); //
    
AssertTrue(
    F_SafeBPCompare(stSafer, stNotSoSafe),
    'Rate eval is broken (True)'); 

AssertFalse(
    F_SafeBPCompare(stNotSoSafe, stSafer),
    'Rate eval is broken (False)');
TEST_FINISHED();
    
//Pulse energy
TEST('BPComparisonPulseEnergy');
stSafer := F_SetBeamParams(
    0, 
    1, //
    16#FFFF,
    1,
    PMPS_GVL.DUMMY_AUX_ATT_ARRAY);

stNotSoSafe := F_SetBeamParams(
    0, 
    10, //
    16#FFFF,
    1,
    PMPS_GVL.DUMMY_AUX_ATT_ARRAY); 
    
AssertTrue(
    F_SafeBPCompare(stSafer, stNotSoSafe),
    'Pulse energy eval is broken (True)'); 

AssertFalse(
    F_SafeBPCompare(stNotSoSafe, stSafer),
    'Pulse energy eval is broken (False)');    
TEST_FINISHED();
    
//Photon energy
//More extensive tests elsewhere
TEST('BPComparisonPhotonEnergy');
stSafer := F_SetBeamParams(
    0, 
    1, 
    2#0000_0000_0000_0010,
    1,
    PMPS_GVL.DUMMY_AUX_ATT_ARRAY);

stNotSoSafe := F_SetBeamParams(
    0, 
    1, 
    2#0000_0000_0000_0110,
    1,
    PMPS_GVL.DUMMY_AUX_ATT_ARRAY);
    
AssertTrue(
    F_SafeBPCompare(stSafer, stNotSoSafe),
    'Photon energy eval is broken (True)'); 

AssertFalse(
    F_SafeBPCompare(stNotSoSafe, stSafer),
    'Photon energy eval is broken (False)');    
TEST_FINISHED();
END_METHOD

END_FUNCTION_BLOCK

// TestComponents/FB_SubsysToArb_Test
{attribute 'call_after_init'}
FUNCTION_BLOCK FB_SubsysToArb_Test EXTENDS TcUnit.FB_TestSuite
VAR_INPUT
END_VAR
VAR_OUTPUT
END_VAR
VAR
END_VAR

BasicFunction();

METHOD BasicFunction
VAR_INPUT
END_VAR
VAR   
    nId    :    DWORD := 1;
    stReq    :    ST_BeamParams := (nTran:=12);
END_VAR
VAR_INST
    fbArbiter    :    FB_Arbiter(1);
    
    fbSubSysToArb : FB_SubSysToArbiter_IO; // Subsystem interface with beamline arbiter PLC
    pBPC : POINTER TO ST_BeamParams_IO;
    
    ioCurrentBP : ST_BeamParams_IO; 
    
    FFO : FB_HardwareFFOutput; // Dummy FFO not important for these tests
    
END_VAR
VAR CONSTANT
    SysID : DWORD := 42;
END_VAR
// This simulates a synchronous cycle between the subsystem and arbiter PLC cycles. Ie. phase is locked, and cycle time is the same. This is not always the case, so these tests should be 
// trusted with a grain of salt.

TEST('Add to arbiter');

IF NOT fbArbiter.CheckRequestInPool(nID) THEN
    AssertTrue(fbArbiter.AddRequest(nId, stReq), 'Arbiter returned false from AddRequest'); // some device asking its local arbiter for some beam parameters
END_IF  
   
TEST_FINISHED();   

///////////////////////////////////////
//Sub system cycle
fbSubSysToArb(Arbiter := fbArbiter, fbFFHWO := FFO);
//END of sub system cycle
///////////////////////////////////////


TEST('Initial Elevation');
AssertTrue(fbSubSysToArb.nRequestCohort = fbSubSysToArb.q_stRequestedBP.nCohortInt, 'ReqCohort and qBP Cohort do not match');
AssertFalse(fbArbiter.xActiveInArbitration, 'Arbiter indicates it is included in arbitration prematurely');
AssertTrue(fbSubSysToArb.nRequestCohort = 1, 'Cohort index should move to 1 with first request');
TEST_FINISHED_NAMED('Initial Elevation');
    
//Ethercat transfer simulation
// Transfer of requested BP to arbiter PLC
// pBPR := ADR(fbArbToSubSys.i_RequestedBP);
// pBPR^ := fbSubSysToArb.q_stRequestedBP;

ioCurrentBP := fbSubSysToArb.q_stRequestedBP;
// NOTE: Setting the returning cohort number to something less than the request cohort number
// will prevent the sub system arbiter FB from considering itself active in arbitration.
// The next set of tests verify this.
ioCurrentBP.nCohortInt := 0;

// Transfer of current BP to sub system PLC
pBPC := ADR(fbSubSysToArb.i_stCurrentBP);
pBPC^ := ioCurrentBP;

///////////////////////////////////////
//Sub system cycle
fbSubSysToArb(Arbiter := fbArbiter, fbFFHWO := FFO);
//END of sub system cycle
///////////////////////////////////////

TEST('Not yet active in arbitration');
AssertTrue(fbSubSysToArb.nActiveCohort = 0, 'Active cohort should still be zero, per ioCurrentBP.nCohortInt setting above.');
AssertFalse(fbArbiter.xActiveInArbitration, 'Arbiter indicates it is included in arbitration prematurely, checkrequest might be broken');
AssertTrue(fbSubSysToArb.nRequestCohort = 1, 'Cohort index should remain at 1 because there have been no additional requests added to the arbiter');
TEST_FINISHED_NAMED('Not yet active in arbitration');

//Ethercat transfer simulation
// Transfer of requested BP to arbiter PLC
// pBPR := ADR(fbArbToSubSys.i_RequestedBP);
// pBPR^ := fbSubSysToArb.q_stRequestedBP;

ioCurrentBP := fbSubSysToArb.q_stRequestedBP;
// NOTE: Now we simulate the FB_ArbiterToSubSys_IO updating the cohort number to the same value as the request cohort, indicating that cohort has been included
ioCurrentBP.nCohortInt := 1;

// Transfer of current BP to sub system PLC
pBPC := ADR(fbSubSysToArb.i_stCurrentBP);
pBPC^ := ioCurrentBP;

///////////////////////////////////////
//Sub system cycle
fbSubSysToArb(Arbiter := fbArbiter, fbFFHWO := FFO);
//END of sub system cycle
///////////////////////////////////////

TEST('Active in arbitration');
AssertTrue(fbSubSysToArb.nActiveCohort = fbSubSysToArb.nRequestCohort, 'Active cohort and request cohort do not match');
AssertTrue(fbArbiter.xActiveInArbitration, 'Arbiter does not indicate it is included in higher arbitration');
TEST_FINISHED_NAMED('Active in arbitration');
END_METHOD

END_FUNCTION_BLOCK

// MAIN
PROGRAM MAIN
VAR
    fbDiffBPTest    :    FB_DiffBP_Test;
    fbBPTMTest    :    FB_BPTM_Test;
    fbSafeBPCompareTest    :    FB_SafeBPCompare_Test;
    //fbevWithinSpecTest    :    FB_evWithinSpec_Test;
    //fbPEWTest    :    FB_PhotonEnergyWatcher_Test;
    fbFFTest    :    FB_FastFault_Test;
    fbArbiterTest    :    FB_Arbiter_Test;
    fbevRangeCalcTest : FB_evRangeCalculator_Test;
    fbSubSysToArbTest : FB_SubsysToArb_Test;
    fbArbToSubSysTest : FB_ArbToSubsys_Test;
END_VAR

TcUnit.RUN();

END_PROGRAM
